{attribute 'qualified_only'}
{attribute 'strict'}
TYPE AutostoreStatus :
(
	UNKNOWN := 0,
	ROTATING	:=1,
	READY	:=2
);
END_TYPE

(* stored: Version 1.1.0.1, ProductVersion 3.1.4024.12
   DUT AutostoreStatus: Id {d6a7edb2-0c30-4660-a148-2e55ffc0e79e} *)
